// Mitsubishi GX Works2 project: Master-Slave-Device-Sensor   PLC: FX3U/FX3UC

PROGRAM MAIN
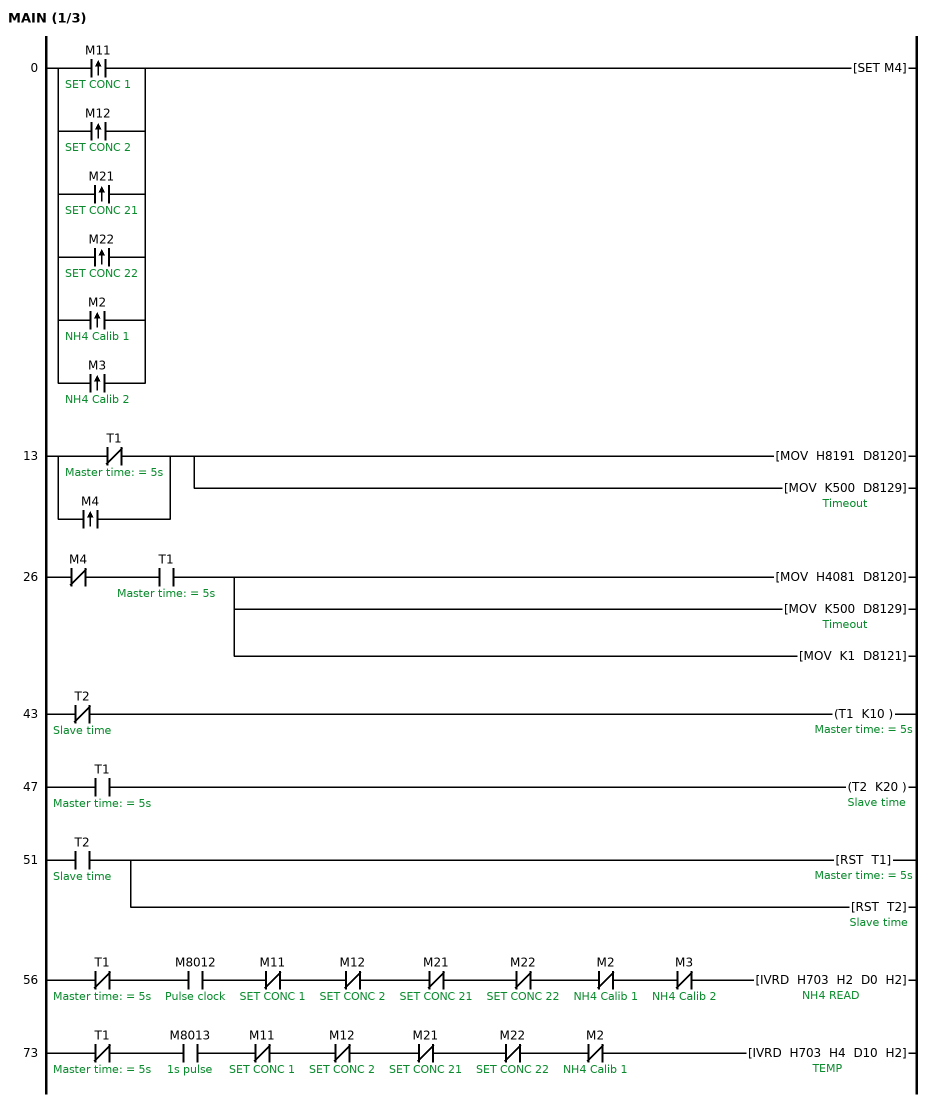
0     LDP     M11  ; SET CONC 1
      ORP     M12  ; SET CONC 2
      ORP     M21  ; SET CONC 21
      ORP     M22  ; SET CONC 22
      ORP     M2  ; NH4 Calib 1
      ORP     M3  ; NH4 Calib 2
      SET     M4
13    LDI     T1  ; Master time: = 5s
      ORP     M4
      MOV     H8191 D8120
      MOV     K500 D8129  ; Timeout
26    LDI     M4
      AND     T1  ; Master time: = 5s
      MOV     H4081 D8120
      MOV     K500 D8129
      MOV     K1 D8121
43    LDI     T2  ; Slave time
      OUT     T1 K10  ; Master time: = 5s
47    LD      T1  ; Master time: = 5s
      OUT     T2 K20  ; Slave time
51    LD      T2  ; Slave time
      RST     T1  ; Master time: = 5s
      RST     T2  ; Slave time
56    LDI     T1  ; Master time: = 5s
      AND     M8012  ; Pulse clock
      ANI     M11  ; SET CONC 1
      ANI     M12  ; SET CONC 2
      ANI     M21  ; SET CONC 21
      ANI     M22  ; SET CONC 22
      ANI     M2  ; NH4 Calib 1
      ANI     M3  ; NH4 Calib 2
      IVRD    H703 H2 D0 H2  ; NH4 READ
73    LDI     T1  ; Master time: = 5s
      AND     M8013  ; 1s pulse
      ANI     M11  ; SET CONC 1
      ANI     M12  ; SET CONC 2
      ANI     M21  ; SET CONC 21
      ANI     M22  ; SET CONC 22
      ANI     M2  ; NH4 Calib 1
      IVRD    H703 H4 D10 H2  ; TEMP
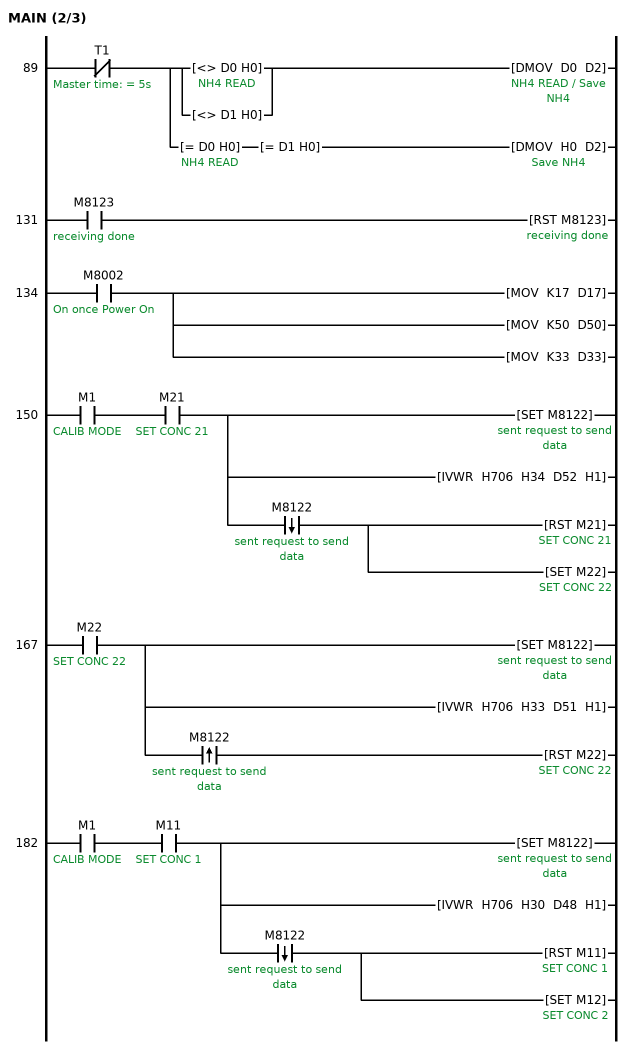
89    LDI     T1  ; Master time: = 5s
      MPS
      LD<>    D0 H0  ; NH4 READ
      OR<>    D1 H0
      ANB
      DMOV    D0 D2  ; Save NH4
      MPP
      AND=    D0 H0  ; NH4 READ
      AND=    D1 H0
      DMOV    H0 D2
131   LD      M8123  ; receiving done
      RST     M8123  ; receiving done
134   LD      M8002  ; On once Power On
      MOV     K17 D17
      MOV     K50 D50
      MOV     K33 D33
150   LD      M1  ; CALIB MODE
      AND     M21  ; SET CONC 21
      SET     M8122  ; sent request to send data
      IVWR    H706 H34 D52 H1
      ANDF    M8122  ; sent request to send data
      RST     M21  ; SET CONC 21
      SET     M22  ; SET CONC 22
167   LD      M22  ; SET CONC 22
      SET     M8122  ; sent request to send data
      IVWR    H706 H33 D51 H1
      ANDP    M8122  ; sent request to send data
      RST     M22  ; SET CONC 22
182   LD      M1  ; CALIB MODE
      AND     M11  ; SET CONC 1
      SET     M8122  ; sent request to send data
      IVWR    H706 H30 D48 H1
      ANDF    M8122  ; sent request to send data
      RST     M11  ; SET CONC 1
      SET     M12  ; SET CONC 2
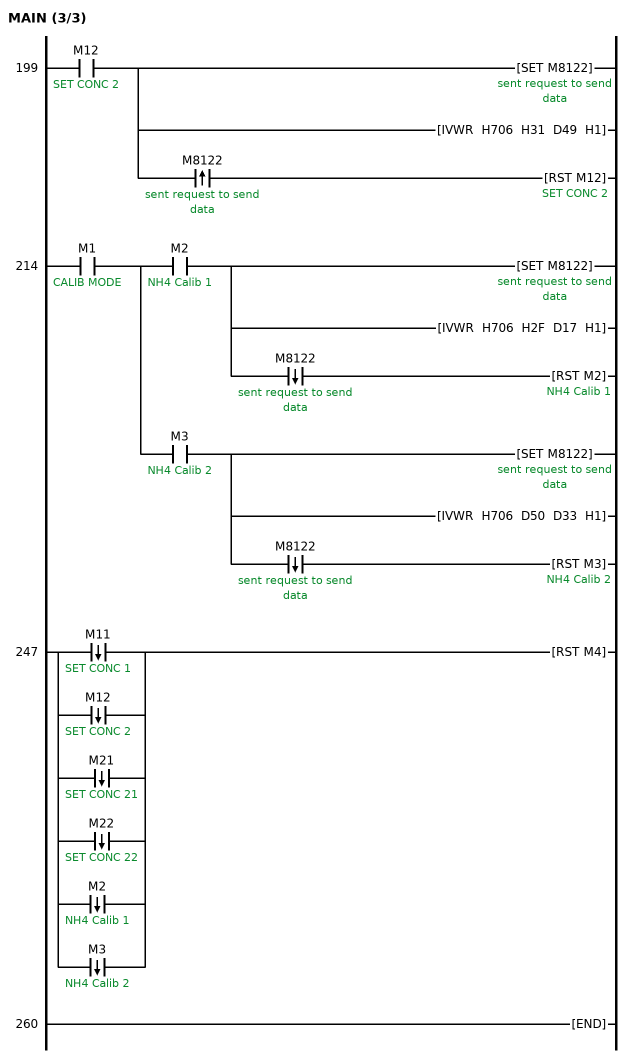
199   LD      M12  ; SET CONC 2
      SET     M8122  ; sent request to send data
      IVWR    H706 H31 D49 H1
      ANDP    M8122  ; sent request to send data
      RST     M12  ; SET CONC 2
214   LD      M1  ; CALIB MODE
      MPS
      AND     M2  ; NH4 Calib 1
      SET     M8122  ; sent request to send data
      IVWR    H706 H2F D17 H1
      ANDF    M8122  ; sent request to send data
      RST     M2  ; NH4 Calib 1
      MPP
      AND     M3  ; NH4 Calib 2
      SET     M8122  ; sent request to send data
      IVWR    H706 D50 D33 H1
      ANDF    M8122  ; sent request to send data
      RST     M3  ; NH4 Calib 2
247   LDF     M11  ; SET CONC 1
      ORF     M12  ; SET CONC 2
      ORF     M21  ; SET CONC 21
      ORF     M22  ; SET CONC 22
      ORF     M2  ; NH4 Calib 1
      ORF     M3  ; NH4 Calib 2
      RST     M4
260   END
END_PROGRAM

// device comments not shown above
M10  ; Master Modce
M13  ; 2 ND REGISTER
C0  ; read param 1
C1  ; change mode
D12  ; MEASURED VALUE pH
D100  ; Float value
D200  ; NH4 Conc. 1: 2mg/L
D202  ; NH4 Conc.2 : 5mg/L
D210  ; heso
D211  ; heso float
D220  ; analog output
D230  ; INT OUT
D240  ; anolog out limited
